PROGRAM MAIN
VAR
END_VAR

P_Modbus_TCP();

END_PROGRAM

(* stored: Version 1.1.0.1, ProductVersion 3.1.4024.6
   POU MAIN: Id {c894818f-67f1-414a-bf39-a157e070adba}, SpecialFunc None *)
